Staubli VAL3: toLowercase.pgx

public program toLowercase(string x_sInput, string& x_sResult)
  local num l_nElement
begin
  x_sResult = ""

  for l_nElement=0 to len(x_sInput)-1
    x_sResult=x_sResult+chr(sel(asc(x_sInput,l_nElement)<65 or asc(x_sInput,l_nElement)>90,asc(x_sInput,l_nElement),asc(x_sInput,l_nElement)+32))
  endFor

end
